TYPE DEV_Sensor_stOutput :
STRUCT
	Abort : BOOL;
	Detecting : BOOL;
END_STRUCT
END_TYPE

(* stored: Version 1.1.0.1, ProductVersion 3.1.4024.6
   DUT DEV_Sensor_stOutput: Id {da2431cc-4b6b-431e-bce4-0bf31de5b949} *)
